Staubli VAL3: HexToDec.pgx

public program HexToDec(string x_sHex, num& x_nDecimal)
  local num l_nIndex
  local num l_nResult
  local bool l_bIsHex
begin

  //upgrade: trim the input string!

  l_bIsHex=false
  call isHexadecimal(x_sHex, l_bIsHex)

  if l_bIsHex
    for l_nIndex=len(x_sHex)-1 to 0 step-1
      l_nResult = l_nResult + (nHex2DecSymbols[mid(x_sHex, 1, l_nIndex)]*power(16, len(x_sHex)-l_nIndex-1))
    endFor
    x_nDecimal = l_nResult
  else
    logMsg("Binary->HexToDec: wrong input format")
  endIf

end
